// TIA Portal project "ExamenSergioZulueta" (V15.1)

(* hardware
DEVICE "S7-1200 station_1"  S7-1200 Station
   slot 0: "Rack_0"  S7-1200 Rack  Rack  V1.0
   slot 1: "PLC_1"  CPU 1214C AC/DC/Rly  6ES7 214-1BG40-0XB0  V4.0
   slot 3: "AQ 1x12BIT_1"  AQ1 signal board  6ES7 232-4HA30-0XB0  V1.0
*)

// ===== PLC "PLC_1"  CPU 1214C AC/DC/Rly =====

VAR_GLOBAL   // PLC tag table "Tabla de variables estándar"
   "Etapa0" AT %M16.0 : Bool;
   "Etapa1" AT %M16.1 : Bool;
   "Etapa2" AT %M16.2 : Bool;
   "Etapa3" AT %M16.3 : Bool;
   "M" AT %I0.0 : Bool;
   "PP" AT %I0.1 : Bool;
   "B0" AT %I0.4 : Bool;
   "B1" AT %I0.5 : Bool;
   "C+" AT %Q0.0 : Bool;
   "C-" AT %Q0.1 : Bool;
   "SEÑALvariador" AT %Q0.2 : Bool;
   "Tag_1" AT %MD70 : DWord;
   "Tag_2" AT %MD74 : Real;
   "Tag_3" AT %QW80 : Word;
   "marcaparo" AT %M19.0 : Bool;
END_VAR

// folder: System blocks/Program resources

DATA_BLOCK "Temporizador1"   // DB1
{ S7_Optimized_Access := 'TRUE' }
AUTHOR : Simatic
FAMILY : IEC
NAME : IEC_TMR
VERSION : 1.0
// stored: InstanceOfName IEC_TIMER
"IEC_TIMER"
BEGIN
END_DATA_BLOCK

DATA_BLOCK "Temporizador2"   // DB2
{ S7_Optimized_Access := 'TRUE' }
AUTHOR : Simatic
FAMILY : IEC
NAME : IEC_TMR
VERSION : 1.0
// stored: InstanceOfName IEC_TIMER
"IEC_TIMER"
BEGIN
END_DATA_BLOCK

// folder: (top level)

FUNCTION "Grafcet" : Void   // FC1, LAD
{ S7_Optimized_Access := 'TRUE' }
VERSION : 0.1
   VAR_TEMP
      marcaparo : Bool;
   END_VAR
BEGIN

REGION Network 1
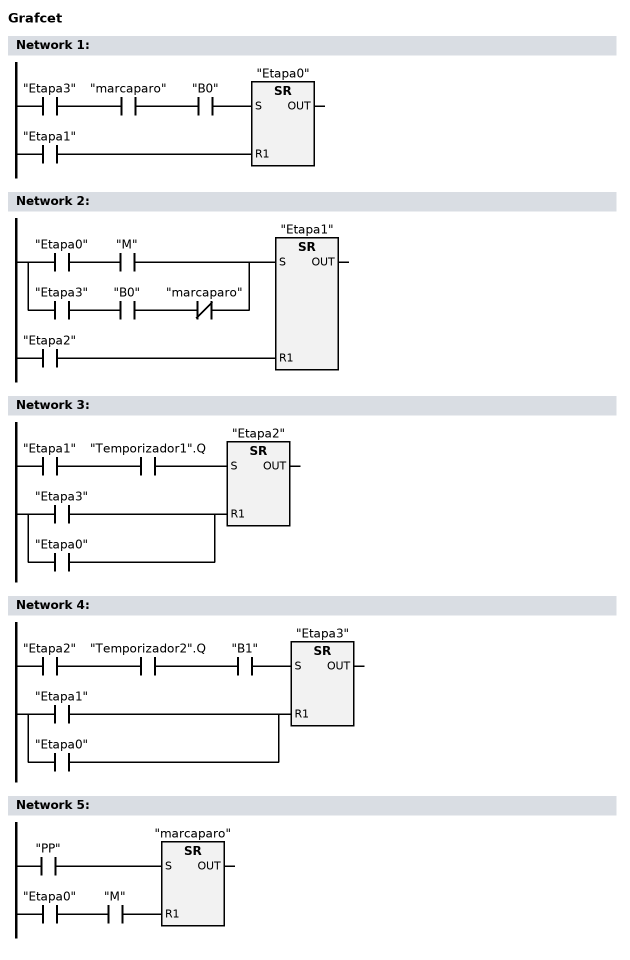
   RUNG wire#powerrail
      Contact( "Etapa3" )
      Contact( "marcaparo" )
      Contact( "B0" )
      S_SR(operand := "Etapa0", r1 := wire#w1)
   END_RUNG
   RUNG wire#powerrail
      Contact( "Etapa1" )
   END_RUNG wire#w1
   // the same network as SCL:
   IF "Etapa3" AND "marcaparo" AND "B0" THEN
       "Etapa0" := TRUE;   // SR flip-flop
   END_IF;
   IF "Etapa1" THEN "Etapa0" := FALSE; END_IF;
END_REGION

REGION Network 2
   RUNG wire#powerrail
      Contact( "Etapa0" )
      Contact( "M" )
      wire#w1
      S_SR(operand := "Etapa1", r1 := wire#w2)
   END_RUNG
   RUNG wire#powerrail
      Contact( "Etapa3" )
      Contact( "B0" )
      I_Contact( "marcaparo" )
   END_RUNG wire#w1
   RUNG wire#powerrail
      Contact( "Etapa2" )
   END_RUNG wire#w2
   // the same network as SCL:
   IF ("Etapa0" AND "M") OR ("Etapa3" AND "B0" AND NOT "marcaparo") THEN
       "Etapa1" := TRUE;   // SR flip-flop
   END_IF;
   IF "Etapa2" THEN "Etapa1" := FALSE; END_IF;
END_REGION

REGION Network 3
   RUNG wire#powerrail
      Contact( "Etapa1" )
      Contact( "Temporizador1".Q )
      S_SR(operand := "Etapa2", r1 := wire#w1)
   END_RUNG
   RUNG wire#powerrail
      Contact( "Etapa3" )
   END_RUNG wire#w1
   RUNG wire#powerrail
      Contact( "Etapa0" )
   END_RUNG wire#w1
   // the same network as SCL:
   IF "Etapa1" AND "Temporizador1".Q THEN
       "Etapa2" := TRUE;   // SR flip-flop
   END_IF;
   IF "Etapa3" OR "Etapa0" THEN "Etapa2" := FALSE; END_IF;
END_REGION

REGION Network 4
   RUNG wire#powerrail
      Contact( "Etapa2" )
      Contact( "Temporizador2".Q )
      Contact( "B1" )
      S_SR(operand := "Etapa3", r1 := wire#w1)
   END_RUNG
   RUNG wire#powerrail
      Contact( "Etapa1" )
   END_RUNG wire#w1
   RUNG wire#powerrail
      Contact( "Etapa0" )
   END_RUNG wire#w1
   // the same network as SCL:
   IF "Etapa2" AND "Temporizador2".Q AND "B1" THEN
       "Etapa3" := TRUE;   // SR flip-flop
   END_IF;
   IF "Etapa1" OR "Etapa0" THEN "Etapa3" := FALSE; END_IF;
END_REGION

REGION Network 5
   RUNG wire#powerrail
      Contact( "PP" )
      S_SR(operand := "marcaparo", r1 := wire#w1)
   END_RUNG
   RUNG wire#powerrail
      Contact( "Etapa0" )
      Contact( "M" )
   END_RUNG wire#w1
   // the same network as SCL:
   IF "PP" THEN
       "marcaparo" := TRUE;   // SR flip-flop
   END_IF;
   IF "Etapa0" AND "M" THEN "marcaparo" := FALSE; END_IF;
END_REGION
END_FUNCTION

FUNCTION "temporizadores" : Void   // FC2, LAD
{ S7_Optimized_Access := 'TRUE' }
VERSION : 0.1
BEGIN

REGION Network 1
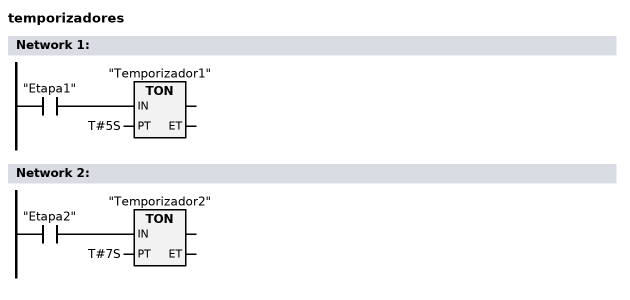
   "Temporizador1".TON(IN := "Etapa1", PT := T#5S);
END_REGION

REGION Network 2
   "Temporizador2".TON(IN := "Etapa2", PT := T#7S);
END_REGION
END_FUNCTION

FUNCTION "Salidas" : Void   // FC3, LAD
{ S7_Optimized_Access := 'TRUE' }
VERSION : 0.1
BEGIN

REGION Network 1
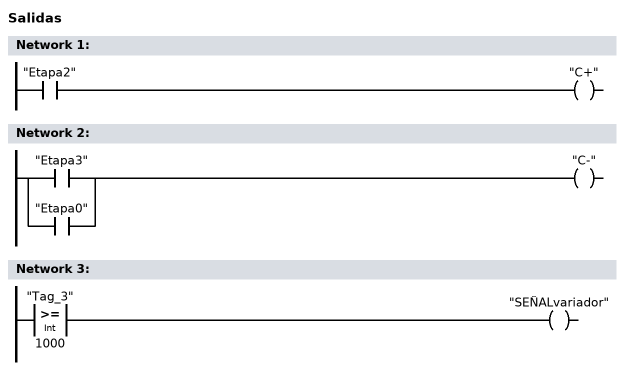
   RUNG wire#powerrail
      Contact( "Etapa2" )
      Coil( "C+" )
   END_RUNG
   // the same network as SCL:
   "C+" := "Etapa2";
END_REGION

REGION Network 2
   RUNG wire#powerrail
      Contact( "Etapa3" )
      wire#w1
      Coil( "C-" )
   END_RUNG
   RUNG wire#powerrail
      Contact( "Etapa0" )
   END_RUNG wire#w1
   // the same network as SCL:
   "C-" := "Etapa3" OR "Etapa0";
END_REGION

REGION Network 3
   RUNG wire#powerrail
      { S7_Templates := "SrcType := Int" } GE_Contact(in1 := "Tag_3", in2 := 1000)
      Coil( "SEÑALvariador" )
   END_RUNG
   // the same network as SCL:
   "SEÑALvariador" := "Tag_3" >= 1000;
END_REGION
END_FUNCTION

FUNCTION "variador" : Void   // FC4, LAD
{ S7_Optimized_Access := 'TRUE' }
VERSION : 0.1
BEGIN

REGION Network 1
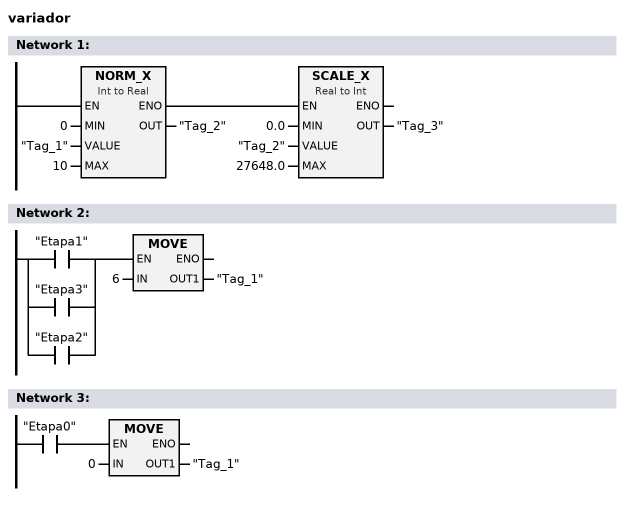
   RUNG wire#powerrail
      { S7_Templates := "[SrcType := Int, DestType := Real]" } Normalize(min := 0, value := "Tag_1", max := 10, out => "Tag_2")
      { S7_Templates := "[SrcType := Real, DestType := Int]" } Scale(min := 0.0, value := "Tag_2", max := 27648.0, out => "Tag_3")
   END_RUNG
   // the same network as SCL:
   "Tag_2" := NORM_X(MIN := 0, VALUE := "Tag_1", MAX := 10);
   "Tag_3" := SCALE_X(MIN := 0.0, VALUE := "Tag_2", MAX := 27648.0);
END_REGION

REGION Network 2
   RUNG wire#powerrail
      Contact( "Etapa1" )
      wire#w1
      Move(in := 6, out1 => "Tag_1")
   END_RUNG
   RUNG wire#powerrail
      Contact( "Etapa3" )
   END_RUNG wire#w1
   RUNG wire#powerrail
      Contact( "Etapa2" )
   END_RUNG wire#w1
   // the same network as SCL:
   IF "Etapa1" OR "Etapa3" OR "Etapa2" THEN "Tag_1" := 6; END_IF;
END_REGION

REGION Network 3
   RUNG wire#powerrail
      Contact( "Etapa0" )
      Move(in := 0, out1 => "Tag_1")
   END_RUNG
   // the same network as SCL:
   IF "Etapa0" THEN "Tag_1" := 0; END_IF;
END_REGION
END_FUNCTION

ORGANIZATION_BLOCK "Main"   // OB1, LAD, ProgramCycle
TITLE = "Main Program Sweep (Cycle)"
{ S7_Optimized_Access := 'TRUE' }
VERSION : 0.1
   VAR_INPUT
      Initial_Call : Bool;   // Initial call of this OB
      Remanence : Bool;   // =True, if remanent data are available
   END_VAR
BEGIN

REGION Network 1
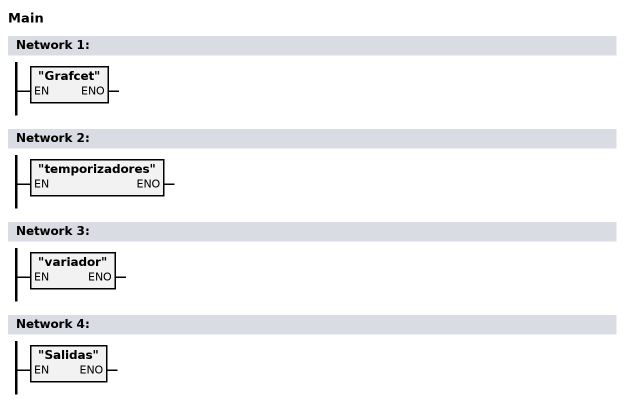
   RUNG wire#powerrail
      "Grafcet"()
   END_RUNG
   // the same network as SCL:
   "Grafcet"();
END_REGION

REGION Network 2
   RUNG wire#powerrail
      "temporizadores"()
   END_RUNG
   // the same network as SCL:
   "temporizadores"();
END_REGION

REGION Network 3
   RUNG wire#powerrail
      "variador"()
   END_RUNG
   // the same network as SCL:
   "variador"();
END_REGION

REGION Network 4
   RUNG wire#powerrail
      "Salidas"()
   END_RUNG
   // the same network as SCL:
   "Salidas"();
END_REGION
END_ORGANIZATION_BLOCK

ORGANIZATION_BLOCK "Startup"   // OB100, LAD, Startup
TITLE = "Complete Restart"
{ S7_Optimized_Access := 'TRUE' }
VERSION : 0.1
   VAR_INPUT
      LostRetentive : Bool;   // True if retentive data are lost
      LostRTC : Bool;   // True if date and time are lost
   END_VAR
BEGIN

REGION Network 1
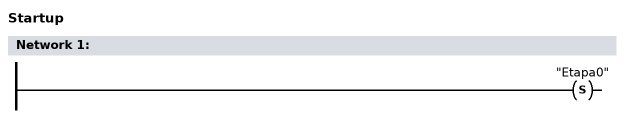
   RUNG wire#powerrail
      S_Coil( "Etapa0" )
   END_RUNG
   // the same network as SCL:
   "Etapa0" := TRUE;
END_REGION
END_ORGANIZATION_BLOCK